// TIA Portal V20 export
FUNCTION_BLOCK "LER_BrakeTest"   // FB179, LAD
// stored: Access Published, MemoryReserve 100, SetENOAutomatically false
   VAR_INPUT
      EnableManualCmds : Bool;
      mcRun : Bool;
      allDoorsOK : Bool;
      all_BrakeTest : "LER_typeBrakeTestUnitCommands";
      statUnitStatus : "LAF_typeUnitStatus";
      hardwareId : HW_IO;
   END_VAR
   VAR_IN_OUT
      BrakeTestControlNoeds : "LER_typeBrakeTestEmControlNodes";
      axis_ControlNode : "LBC_typeAxis64PosControlNode";
      HmiBrakeTestControlNoeds : "LER_typeBrakeTestEmInterface";
   END_VAR
   VAR
      statTonTime { S7_SetPoint := 'True'} : Array[0..10] of TON_TIME;
      statPulse { S7_SetPoint := 'True'} : Array[0..10] of Bool;
      instLDrv701Control { S7_SetPoint := 'True'} : "LDrvSafe_SinaTlg701Control";
      instLDrv701Status { S7_SetPoint := 'True'} : "LDrvSafe_SinaTlg701Status";
   END_VAR
   VAR_TEMP   // added for the SCL form of the ladder/FBD networks
      _w1 : Bool;
      _w2 : Bool;
      _w3 : Bool;
      _w4 : Bool;
   END_VAR
BEGIN

REGION Network 2: Error Check
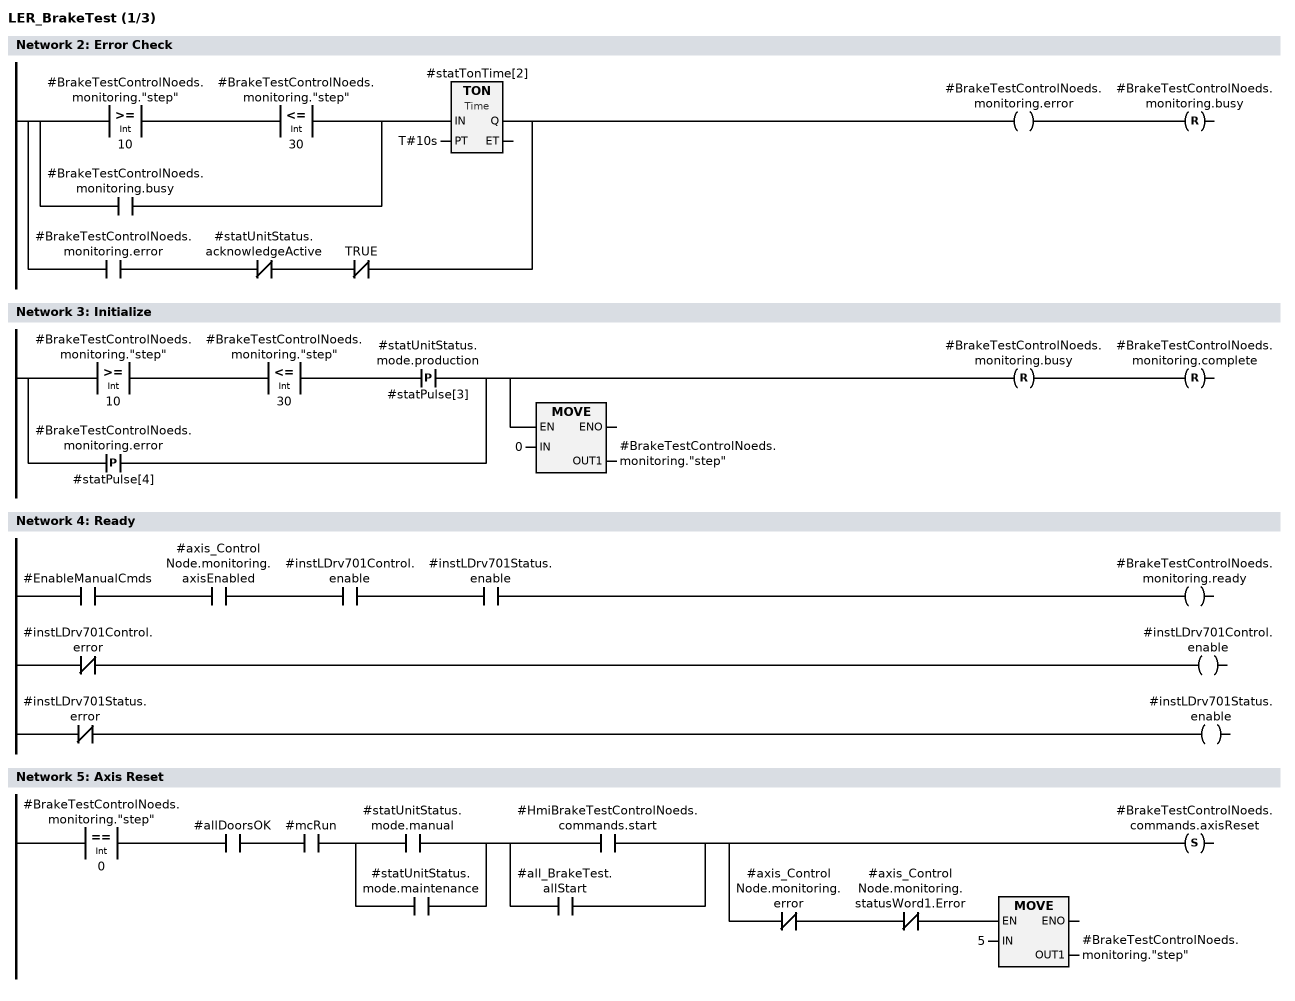
   RUNG wire#powerrail
      { S7_Templates := "SrcType := Int" } GE_Contact(in1 := #BrakeTestControlNoeds.monitoring."step", in2 := 10)
      { S7_Templates := "SrcType := Int" } LE_Contact(in1 := #BrakeTestControlNoeds.monitoring."step", in2 := 30)
      wire#w1
      { S7_Templates := "time_type := Time" } #statTonTime[2].TON(pt := T#10s, et =>)
      wire#w2
      Coil( #BrakeTestControlNoeds.monitoring.error )
      R_Coil( #BrakeTestControlNoeds.monitoring.busy )
   END_RUNG
   RUNG wire#powerrail
      Contact( #BrakeTestControlNoeds.monitoring.busy )
   END_RUNG wire#w1
   RUNG wire#powerrail
      Contact( #BrakeTestControlNoeds.monitoring.error )
      I_Contact( #statUnitStatus.acknowledgeActive )
      I_Contact( TRUE )
   END_RUNG wire#w2
   // the same network as SCL:
   #statTonTime[2].TON(IN := ((#BrakeTestControlNoeds.monitoring."step" >= 10) AND (#BrakeTestControlNoeds.monitoring."step" <= 30)) OR #BrakeTestControlNoeds.monitoring.busy,
                       PT := T#10s);
   #BrakeTestControlNoeds.monitoring.error := #statTonTime[2].Q OR (#BrakeTestControlNoeds.monitoring.error AND NOT #statUnitStatus.acknowledgeActive AND NOT TRUE);
   IF #BrakeTestControlNoeds.monitoring.error THEN #BrakeTestControlNoeds.monitoring.busy := FALSE; END_IF;
END_REGION

REGION Network 3: Initialize
   RUNG wire#powerrail
      { S7_Templates := "SrcType := Int" } GE_Contact(in1 := #BrakeTestControlNoeds.monitoring."step", in2 := 10)
      { S7_Templates := "SrcType := Int" } LE_Contact(in1 := #BrakeTestControlNoeds.monitoring."step", in2 := 30)
      P_Contact(operand := #statUnitStatus.mode.production, bit := #statPulse[3])
      wire#w1
      R_Coil( #BrakeTestControlNoeds.monitoring.busy )
      R_Coil( #BrakeTestControlNoeds.monitoring.complete )
   END_RUNG
   RUNG wire#powerrail
      P_Contact(operand := #BrakeTestControlNoeds.monitoring.error, bit := #statPulse[4])
   END_RUNG wire#w1
   RUNG wire#w1
      Move(in := 0, out1 => #BrakeTestControlNoeds.monitoring."step")
   END_RUNG
   // the same network as SCL:
   #_w1 := (#BrakeTestControlNoeds.monitoring."step" >= 10) AND (#BrakeTestControlNoeds.monitoring."step" <= 30) AND #statUnitStatus.mode.production AND NOT #statPulse[3];   // rising edge of #statUnitStatus.mode.production
   #statPulse[3] := #statUnitStatus.mode.production;
   #_w2 := #BrakeTestControlNoeds.monitoring.error AND NOT #statPulse[4];   // rising edge of #BrakeTestControlNoeds.monitoring.error
   #statPulse[4] := #BrakeTestControlNoeds.monitoring.error;
   IF #_w1 OR #_w2 THEN
       #BrakeTestControlNoeds.monitoring.busy := FALSE;
       #BrakeTestControlNoeds.monitoring.complete := FALSE;
       #BrakeTestControlNoeds.monitoring."step" := 0;
   END_IF;
END_REGION

REGION Network 4: Ready
   RUNG wire#powerrail
      Contact( #EnableManualCmds )
      Contact( #axis_ControlNode.monitoring.axisEnabled )
      Contact( #instLDrv701Control.enable )
      Contact( #instLDrv701Status.enable )
      Coil( #BrakeTestControlNoeds.monitoring.ready )
   END_RUNG
   RUNG wire#powerrail
      I_Contact( #instLDrv701Control.error )
      Coil( #instLDrv701Control.enable )
   END_RUNG
   RUNG wire#powerrail
      I_Contact( #instLDrv701Status.error )
      Coil( #instLDrv701Status.enable )
   END_RUNG
   // the same network as SCL:
   #BrakeTestControlNoeds.monitoring.ready := #EnableManualCmds AND #axis_ControlNode.monitoring.axisEnabled AND #instLDrv701Control.enable AND #instLDrv701Status.enable;
   #instLDrv701Control.enable := NOT #instLDrv701Control.error;
   #instLDrv701Status.enable := NOT #instLDrv701Status.error;
END_REGION

REGION Network 5: Axis Reset
   RUNG wire#powerrail
      { S7_Templates := "SrcType := Int" } EQ_Contact(in1 := #BrakeTestControlNoeds.monitoring."step", in2 := 0)
      Contact( #allDoorsOK )
      Contact( #mcRun )
      wire#w1
      Contact( #statUnitStatus.mode.manual )
      wire#w2
      Contact( #HmiBrakeTestControlNoeds.commands.start )
      wire#w3
      S_Coil( #BrakeTestControlNoeds.commands.axisReset )
   END_RUNG
   RUNG wire#w1
      Contact( #statUnitStatus.mode.maintenance )
   END_RUNG wire#w2
   RUNG wire#w2
      Contact( #all_BrakeTest.allStart )
   END_RUNG wire#w3
   RUNG wire#w3
      I_Contact( #axis_ControlNode.monitoring.error )
      I_Contact( #axis_ControlNode.monitoring.statusWord1.Error )
      Move(in := 5, out1 => #BrakeTestControlNoeds.monitoring."step")
   END_RUNG
   // the same network as SCL:
   #_w1 := (#BrakeTestControlNoeds.monitoring."step" = 0) AND #allDoorsOK AND #mcRun AND (#statUnitStatus.mode.manual OR #statUnitStatus.mode.maintenance) AND (#HmiBrakeTestControlNoeds.commands.start OR #all_BrakeTest.allStart);
   IF #_w1 THEN #BrakeTestControlNoeds.commands.axisReset := TRUE; END_IF;
   IF #_w1 AND NOT #axis_ControlNode.monitoring.error AND NOT #axis_ControlNode.monitoring.statusWord1.Error THEN
       #BrakeTestControlNoeds.monitoring."step" := 5;
   END_IF;
END_REGION

REGION Network 6: Commands
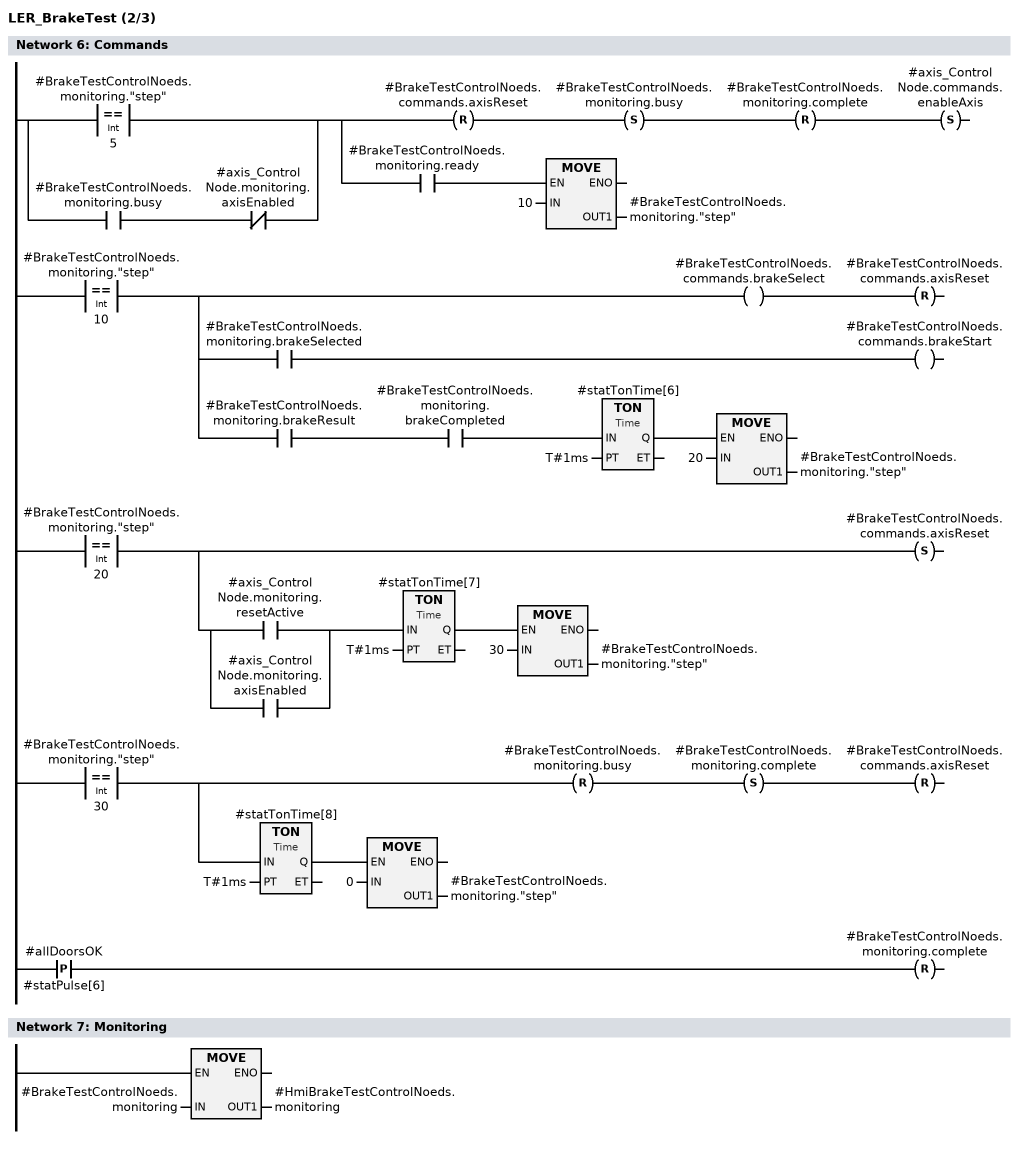
   RUNG wire#powerrail
      { S7_Templates := "SrcType := Int" } EQ_Contact(in1 := #BrakeTestControlNoeds.monitoring."step", in2 := 5)
      wire#w1
      R_Coil( #BrakeTestControlNoeds.commands.axisReset )
      S_Coil( #BrakeTestControlNoeds.monitoring.busy )
      R_Coil( #BrakeTestControlNoeds.monitoring.complete )
      S_Coil( #axis_ControlNode.commands.enableAxis )
   END_RUNG
   RUNG wire#powerrail
      Contact( #BrakeTestControlNoeds.monitoring.busy )
      I_Contact( #axis_ControlNode.monitoring.axisEnabled )
   END_RUNG wire#w1
   RUNG wire#w1
      Contact( #BrakeTestControlNoeds.monitoring.ready )
      Move(in := 10, out1 => #BrakeTestControlNoeds.monitoring."step")
   END_RUNG
   RUNG wire#powerrail
      { S7_Templates := "SrcType := Int" } EQ_Contact(in1 := #BrakeTestControlNoeds.monitoring."step", in2 := 10)
      wire#w2
      Coil( #BrakeTestControlNoeds.commands.brakeSelect )
      R_Coil( #BrakeTestControlNoeds.commands.axisReset )
   END_RUNG
   RUNG wire#w2
      Contact( #BrakeTestControlNoeds.monitoring.brakeSelected )
      Coil( #BrakeTestControlNoeds.commands.brakeStart )
   END_RUNG
   RUNG wire#w2
      Contact( #BrakeTestControlNoeds.monitoring.brakeResult )
      Contact( #BrakeTestControlNoeds.monitoring.brakeCompleted )
      { S7_Templates := "time_type := Time" } #statTonTime[6].TON(pt := T#1ms, et =>)
      Move(in := 20, out1 => #BrakeTestControlNoeds.monitoring."step")
   END_RUNG
   RUNG wire#powerrail
      { S7_Templates := "SrcType := Int" } EQ_Contact(in1 := #BrakeTestControlNoeds.monitoring."step", in2 := 20)
      wire#w3
      S_Coil( #BrakeTestControlNoeds.commands.axisReset )
   END_RUNG
   RUNG wire#w3
      Contact( #axis_ControlNode.monitoring.resetActive )
      wire#w4
      { S7_Templates := "time_type := Time" } #statTonTime[7].TON(pt := T#1ms, et =>)
      Move(in := 30, out1 => #BrakeTestControlNoeds.monitoring."step")
   END_RUNG
   RUNG wire#w3
      Contact( #axis_ControlNode.monitoring.axisEnabled )
   END_RUNG wire#w4
   RUNG wire#powerrail
      { S7_Templates := "SrcType := Int" } EQ_Contact(in1 := #BrakeTestControlNoeds.monitoring."step", in2 := 30)
      wire#w5
      R_Coil( #BrakeTestControlNoeds.monitoring.busy )
      S_Coil( #BrakeTestControlNoeds.monitoring.complete )
      R_Coil( #BrakeTestControlNoeds.commands.axisReset )
   END_RUNG
   RUNG wire#w5
      { S7_Templates := "time_type := Time" } #statTonTime[8].TON(pt := T#1ms, et =>)
      Move(in := 0, out1 => #BrakeTestControlNoeds.monitoring."step")
   END_RUNG
   RUNG wire#powerrail
      P_Contact(operand := #allDoorsOK, bit := #statPulse[6])
      R_Coil( #BrakeTestControlNoeds.monitoring.complete )
   END_RUNG
   // the same network as SCL:
   #_w1 := (#BrakeTestControlNoeds.monitoring."step" = 5) OR (#BrakeTestControlNoeds.monitoring.busy AND NOT #axis_ControlNode.monitoring.axisEnabled);
   IF #_w1 THEN
       #BrakeTestControlNoeds.commands.axisReset := FALSE;
       #BrakeTestControlNoeds.monitoring.busy := TRUE;
       #BrakeTestControlNoeds.monitoring.complete := FALSE;
       #axis_ControlNode.commands.enableAxis := TRUE;
   END_IF;
   IF #_w1 AND #BrakeTestControlNoeds.monitoring.ready THEN
       #BrakeTestControlNoeds.monitoring."step" := 10;
   END_IF;
   #BrakeTestControlNoeds.commands.brakeSelect := #BrakeTestControlNoeds.monitoring."step" = 10;
   IF #BrakeTestControlNoeds.commands.brakeSelect THEN
       #BrakeTestControlNoeds.commands.axisReset := FALSE;
   END_IF;
   #BrakeTestControlNoeds.commands.brakeStart := #BrakeTestControlNoeds.commands.brakeSelect AND #BrakeTestControlNoeds.monitoring.brakeSelected;
   #statTonTime[6].TON(IN := #BrakeTestControlNoeds.commands.brakeSelect AND #BrakeTestControlNoeds.monitoring.brakeResult AND #BrakeTestControlNoeds.monitoring.brakeCompleted,
                       PT := T#1ms);
   IF #statTonTime[6].Q THEN #BrakeTestControlNoeds.monitoring."step" := 20; END_IF;
   #_w2 := #BrakeTestControlNoeds.monitoring."step" = 20;
   IF #_w2 THEN #BrakeTestControlNoeds.commands.axisReset := TRUE; END_IF;
   #statTonTime[7].TON(IN := #_w2 AND (#axis_ControlNode.monitoring.resetActive OR #axis_ControlNode.monitoring.axisEnabled),
                       PT := T#1ms);
   IF #statTonTime[7].Q THEN #BrakeTestControlNoeds.monitoring."step" := 30; END_IF;
   #_w3 := #BrakeTestControlNoeds.monitoring."step" = 30;
   IF #_w3 THEN
       #BrakeTestControlNoeds.monitoring.busy := FALSE;
       #BrakeTestControlNoeds.monitoring.complete := TRUE;
       #BrakeTestControlNoeds.commands.axisReset := FALSE;
   END_IF;
   #statTonTime[8].TON(IN := #_w3, PT := T#1ms);
   IF #statTonTime[8].Q THEN #BrakeTestControlNoeds.monitoring."step" := 0; END_IF;
   #_w4 := #allDoorsOK AND NOT #statPulse[6];   // rising edge of #allDoorsOK
   #statPulse[6] := #allDoorsOK;
   IF #_w4 THEN #BrakeTestControlNoeds.monitoring.complete := FALSE; END_IF;
END_REGION

REGION Network 7: Monitoring
   RUNG wire#powerrail
      Move(in := #BrakeTestControlNoeds.monitoring, out1 => #HmiBrakeTestControlNoeds.monitoring)
   END_RUNG
   // the same network as SCL:
   #HmiBrakeTestControlNoeds.monitoring := #BrakeTestControlNoeds.monitoring;
END_REGION

REGION Network 8: Call Telegram 701
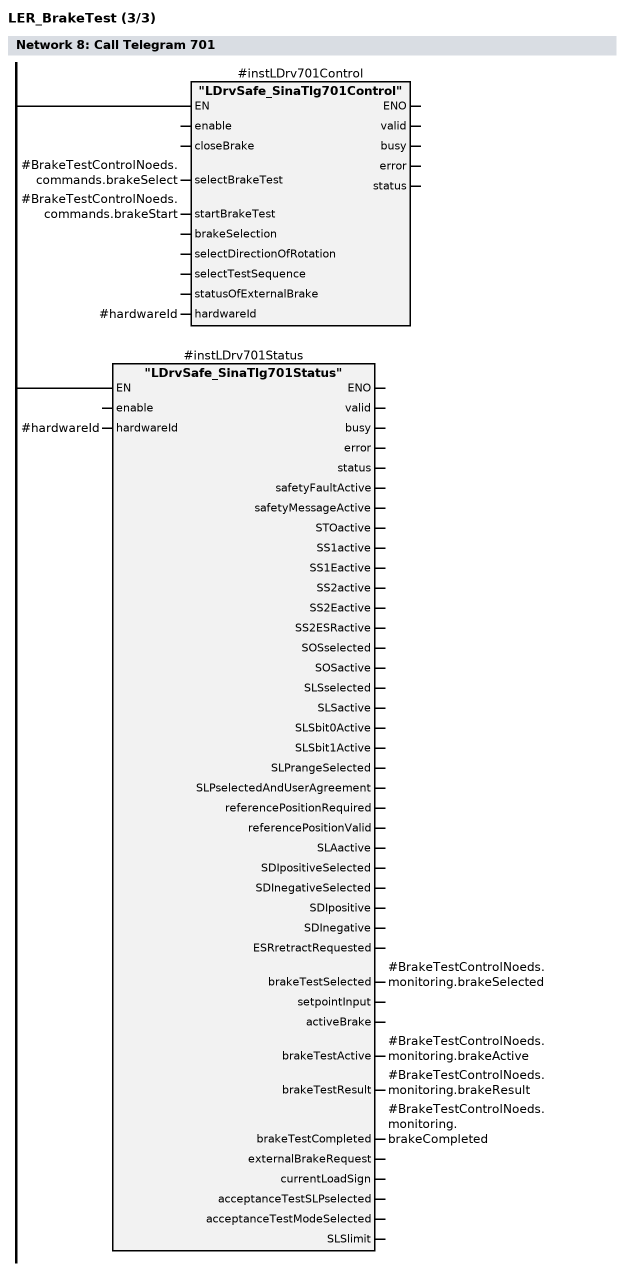
   RUNG wire#powerrail
      #instLDrv701Control(enable :=, closeBrake :=, selectBrakeTest := #BrakeTestControlNoeds.commands.brakeSelect, startBrakeTest := #BrakeTestControlNoeds.commands.brakeStart, brakeSelection :=, selectDirectionOfRotation :=, selectTestSequence :=, statusOfExternalBrake :=, hardwareId := #hardwareId, valid =>, busy =>, error =>, status =>)
   END_RUNG
   RUNG wire#powerrail
      #instLDrv701Status(enable :=, hardwareId := #hardwareId, valid =>, busy =>, error =>, status =>, safetyFaultActive =>, safetyMessageActive =>, STOactive =>, SS1active =>, SS1Eactive =>, SS2active =>, SS2Eactive =>, SS2ESRactive =>, SOSselected =>, SOSactive =>, SLSselected =>, SLSactive =>, SLSbit0Active =>, SLSbit1Active =>, SLPrangeSelected =>, SLPselectedAndUserAgreement =>, referencePositionRequired =>, referencePositionValid =>, SLAactive =>, SDIpositiveSelected =>, SDInegativeSelected =>, SDIpositive =>, SDInegative =>, ESRretractRequested =>, brakeTestSelected => #BrakeTestControlNoeds.monitoring.brakeSelected, setpointInput =>, activeBrake =>, brakeTestActive => #BrakeTestControlNoeds.monitoring.brakeActive, brakeTestResult => #BrakeTestControlNoeds.monitoring.brakeResult, brakeTestCompleted => #BrakeTestControlNoeds.monitoring.brakeCompleted, externalBrakeRequest =>, currentLoadSign =>, acceptanceTestSLPselected =>, acceptanceTestModeSelected =>, SLSlimit =>)
   END_RUNG
   // the same network as SCL:
   #instLDrv701Control(selectBrakeTest := #BrakeTestControlNoeds.commands.brakeSelect,   // "LDrvSafe_SinaTlg701Control"
                       startBrakeTest := #BrakeTestControlNoeds.commands.brakeStart,
                       hardwareId := #hardwareId);
   #instLDrv701Status(hardwareId := #hardwareId,   // "LDrvSafe_SinaTlg701Status"
                      brakeTestSelected => #BrakeTestControlNoeds.monitoring.brakeSelected,
                      brakeTestActive => #BrakeTestControlNoeds.monitoring.brakeActive,
                      brakeTestResult => #BrakeTestControlNoeds.monitoring.brakeResult,
                      brakeTestCompleted => #BrakeTestControlNoeds.monitoring.brakeCompleted);
END_REGION
END_FUNCTION_BLOCK
